# EPICS substitutions: pmc/dls/CS_example.substitutions
file CS_blade_slits.pmc
{pattern
{COORD,PLC,BPLUS,BMINUS,BPMRES,BPOFF,BMMRES,BMOFF,DEFCENTRE,DEFGAP}
{1,    16, 1,    3,     0.001, 0.982,-0.001,-0.65,0,        1000  }
{2,    17, 2,    4,     0.001, 0.632,-0.001,-0.35,0,        1500  }
}
